# EPICS autosave request: ipApp/Db/Rigol_DS1000Z_ChN_settings.req
$(P)$(R)$(CH)Display
$(P)$(R)$(CH)BWLimit
$(P)$(R)$(CH)Coupling
$(P)$(R)$(CH)Invert
$(P)$(R)$(CH)Offset
$(P)$(R)$(CH)Probe
$(P)$(R)$(CH)Scale
